PROGRAM MAIN
VAR
END_VAR

(* 
	GOF 		Separate the construction of a complex object from its representation so that
				the same construction process can create different representations.
*)
P_Builder();

END_PROGRAM

(* stored: Version 1.1.0.1, ProductVersion 3.1.4024.12
   POU MAIN: Id {15e1695a-aab8-4b4f-8888-3359ef891a42}, SpecialFunc None *)
